# EPICS substitutions: ek9000App/Db/EL2001.substitutions
file EL2001.template
{ 	pattern
	{
		TERMINAL,
		DESC1,	ZNAM1,	ONAM1,	PINI1
	}
	{
	}
}
